LIN {X 0,Y 76.368,Z 462.754,A -85,B 0,C 180,E1 -16863.516,E2 -16863.516} C_VEL
LIN {X 0,Y 76.196,Z 460.368,A -85,B 0,C 180,E1 -16851.651,E2 -16851.651} C_VEL
LIN {X 0,Y 77.548,Z 457.672,A -85,B 0,C 180,E1 -16843.095,E2 -16843.095} C_VEL
LIN {X 0,Y 80.04,Z 454.152,A -85,B 0,C 180,E1 -16835.037,E2 -16835.037} C_VEL
LIN {X 0,Y 84.954,Z 448.19,A -85,B 0,C 180,E1 -16825.255,E2 -16825.255} C_VEL
LIN {X 0,Y 90.817,Z 441.616,A -85,B 0,C 180,E1 -16817.713,E2 -16817.713} C_VEL
LIN {X 0,Y 97.828,Z 433.607,A -85,B 0,C 180,E1 -16811.138,E2 -16811.138} C_VEL
LIN {X 0,Y 105.868,Z 423.896,A -85,B 0,C 180,E1 -16805.487,E2 -16805.487} C_VEL
LIN {X 0,Y 112.858,Z 414.711,A -85,B 0,C 180,E1 -16801.582,E2 -16801.582} C_VEL
LIN {X 0,Y 115.371,Z 410.573,A -85,B 0,C 180,E1 -16799.882,E2 -16799.882} C_VEL
LIN {X 0,Y 118.211,Z 403.586,A -85,B 0,C 180,E1 -16796.713,E2 -16796.713} C_VEL
LIN {X 0,Y 121.079,Z 396.289,A -85,B 0,C 180,E1 -16793.8,E2 -16793.8} C_VEL
LIN {X 0,Y 123.45,Z 391.571,A -85,B 0,C 180,E1 -16792.555,E2 -16792.555} C_VEL
LIN {X 0,Y 130.553,Z 378.137,A -85,B 0,C 180,E1 -16790.263,E2 -16790.263} C_VEL
LIN {X 0,Y 134.162,Z 370.217,A -85,B 0,C 180,E1 -16789.189,E2 -16789.189} C_VEL
LIN {X 0,Y 133.423,Z 370.173,A -85,B 0,C 180,E1 -16788.645,E2 -16788.645} C_VEL
LIN {X 0,Y 123.991,Z 379.977,A -85,B 0,C 180,E1 -16786.279,E2 -16786.279} C_VEL
LIN {X 0,Y 117.805,Z 385.302,A -85,B 0,C 180,E1 -16784.146,E2 -16784.146} C_VEL
LIN {X 0,Y 111.854,Z 389.553,A -85,B 0,C 180,E1 -16781.281,E2 -16781.281} C_VEL
LIN {X 0,Y 106.22,Z 394.346,A -85,B 0,C 180,E1 -16778.946,E2 -16778.946} C_VEL
LIN {X 0,Y 101.258,Z 398.024,A -85,B 0,C 180,E1 -16776.156,E2 -16776.156} C_VEL
LIN {X 0,Y 97.039,Z 400.849,A -85,B 0,C 180,E1 -16772.902,E2 -16772.902} C_VEL
LIN {X 0,Y 90.596,Z 405.763,A -85,B 0,C 180,E1 -16767.741,E2 -16767.741} C_VEL
LIN {X 0,Y 84.281,Z 410.653,A -85,B 0,C 180,E1 -16759.486,E2 -16759.486} C_VEL
LIN {X 0,Y 81.446,Z 413.429,A -85,B 0,C 180,E1 -16755.005,E2 -16755.005} C_VEL
LIN {X 0,Y 79.154,Z 416.279,A -85,B 0,C 180,E1 -16747.655,E2 -16747.655} C_VEL
LIN {X 0,Y 76.953,Z 420.193,A -85,B 0,C 180,E1 -16740.002,E2 -16740.002} C_VEL
LIN {X 0,Y 77.191,Z 424.191,A -85,B 0,C 180,E1 -16729.51,E2 -16729.51} C_VEL
LIN {X 0,Y 79.178,Z 430.201,A -85,B 0,C 180,E1 -16716.459,E2 -16716.459} C_VEL
LIN {X 0,Y 82.647,Z 433.114,A -85,B 0,C 180,E1 -16709.323,E2 -16709.323} C_VEL
LIN {X 0,Y 92.152,Z 437.49,A -85,B 0,C 180,E1 -16698.471,E2 -16698.471} C_VEL
LIN {X 0,Y 91.589,Z 439.223,A -85,B 0,C 180,E1 -16696.801,E2 -16696.801} C_VEL
LIN {X 0,Y 83.49,Z 446.528,A -85,B 0,C 180,E1 -16690.749,E2 -16690.749} C_VEL
LIN {X 0,Y 77.128,Z 452.633,A -85,B 0,C 180,E1 -16683.143,E2 -16683.143} C_VEL
LIN {X 0,Y 72.236,Z 458.21,A -85,B 0,C 180,E1 -16672.903,E2 -16672.903} C_VEL
LIN {X 0,Y 69.917,Z 462.377,A -85,B 0,C 180,E1 -16661.598,E2 -16661.598} C_VEL
LIN {X 0,Y 69.61,Z 463.952,A -85,B 0,C 180,E1 -16655.795,E2 -16655.795} C_VEL
LIN {X 0,Y 69.707,Z 465.196,A -85,B 0,C 180,E1 -16650,E2 -16650} C_VEL
LIN {X 0,Y 69.949,Z 466.704,A -85,B 0,C 180,E1 -16638.408,E2 -16638.408} C_VEL
LIN {X 0,Y 72.306,Z 467.097,A -85,B 0,C 180,E1 -16627.121,E2 -16627.121} C_VEL
LIN {X 0,Y 77.196,Z 466.368,A -85,B 0,C 180,E1 -16616.89,E2 -16616.89} C_VEL
LIN {X 0,Y 84.217,Z 464.543,A -85,B 0,C 180,E1 -16608.117,E2 -16608.117} C_VEL
LIN {X 0,Y 92.984,Z 461.628,A -85,B 0,C 180,E1 -16600.902,E2 -16600.902} C_VEL
LIN {X 0,Y 78.146,Z 461.321,A -85,B 0,C 180,E1 -16559.998,E2 -16559.998} C_VEL
LIN {X 0,Y 82.82,Z 461.492,A -85,B 0,C 180,E1 -16545.25,E2 -16545.25} C_VEL
LIN {X 0,Y 86.083,Z 461.662,A -85,B 0,C 180,E1 -16539.043,E2 -16539.043} C_VEL
LIN {X 0,Y 84.24,Z 462.202,A -85,B 0,C 180,E1 -16536.594,E2 -16536.594} C_VEL
LIN {X 0,Y 76.311,Z 463.737,A -85,B 0,C 180,E1 -16525.983,E2 -16525.983} C_VEL
LIN {X 0,Y 72.236,Z 463.873,A -85,B 0,C 180,E1 -16517.072,E2 -16517.072} C_VEL
LIN {X 0,Y 69.528,Z 463.058,A -85,B 0,C 180,E1 -16506.032,E2 -16506.032} C_VEL
LIN {X 0,Y 68.936,Z 460.88,A -85,B 0,C 180,E1 -16493.425,E2 -16493.425} C_VEL
LIN {X 0,Y 70.739,Z 457.451,A -85,B 0,C 180,E1 -16481.461,E2 -16481.461} C_VEL
LIN {X 0,Y 73.551,Z 453.808,A -85,B 0,C 180,E1 -16472.738,E2 -16472.738} C_VEL
LIN {X 0,Y 79.159,Z 447.606,A -85,B 0,C 180,E1 -16462.215,E2 -16462.215} C_VEL
LIN {X 0,Y 85.499,Z 440.957,A -85,B 0,C 180,E1 -16454.505,E2 -16454.505} C_VEL
LIN {X 0,Y 93.156,Z 432.752,A -85,B 0,C 180,E1 -16447.839,E2 -16447.839} C_VEL
LIN {X 0,Y 100.437,Z 424.367,A -85,B 0,C 180,E1 -16442.946,E2 -16442.946} C_VEL
LIN {X 0,Y 108.34,Z 414.448,A -85,B 0,C 180,E1 -16438.738,E2 -16438.738} C_VEL
LIN {X 0,Y 116.635,Z 402.628,A -85,B 0,C 180,E1 -16435.08,E2 -16435.08} C_VEL
LIN {X 0,Y 123.45,Z 391.571,A -85,B 0,C 180,E1 -16432.555,E2 -16432.555} C_VEL
LIN {X 0,Y 123.693,Z 390.413,A -85,B 0,C 180,E1 -16432.047,E2 -16432.047} C_VEL
LIN {X 0,Y 122.96,Z 389.526,A -85,B 0,C 180,E1 -16431.012,E2 -16431.012} C_VEL
LIN {X 0,Y 120.68,Z 389.525,A -85,B 0,C 180,E1 -16429.342,E2 -16429.342} C_VEL
LIN {X 0,Y 117.78,Z 390.583,A -85,B 0,C 180,E1 -16427.744,E2 -16427.744} C_VEL
LIN {X 0,Y 110.801,Z 394.743,A -85,B 0,C 180,E1 -16424.483,E2 -16424.483} C_VEL
LIN {X 0,Y 103.705,Z 399.598,A -85,B 0,C 180,E1 -16421.335,E2 -16421.335} C_VEL
LIN {X 0,Y 97.384,Z 403.751,A -85,B 0,C 180,E1 -16417.839,E2 -16417.839} C_VEL
LIN {X 0,Y 92.834,Z 406.61,A -85,B 0,C 180,E1 -16414.598,E2 -16414.598} C_VEL
LIN {X 0,Y 86.117,Z 411.175,A -85,B 0,C 180,E1 -16409.32,E2 -16409.32} C_VEL
LIN {X 0,Y 80.97,Z 414.622,A -85,B 0,C 180,E1 -16402.993,E2 -16402.993} C_VEL
LIN {X 0,Y 76.41,Z 418.434,A -85,B 0,C 180,E1 -16396.019,E2 -16396.019} C_VEL
LIN {X 0,Y 74.563,Z 420.264,A -85,B 0,C 180,E1 -16390.868,E2 -16390.868} C_VEL
LIN {X 0,Y 71.362,Z 425.036,A -85,B 0,C 180,E1 -16380.002,E2 -16380.002} C_VEL
LIN {X 0,Y 71.472,Z 428.917,A -85,B 0,C 180,E1 -16368.66,E2 -16368.66} C_VEL
LIN {X 0,Y 72.869,Z 433.562,A -85,B 0,C 180,E1 -16357.309,E2 -16357.309} C_VEL
LIN {X 0,Y 77.582,Z 437.267,A -85,B 0,C 180,E1 -16347.078,E2 -16347.078} C_VEL
LIN {X 0,Y 81.006,Z 438.858,A -85,B 0,C 180,E1 -16342.606,E2 -16342.606} C_VEL
LIN {X 0,Y 84.293,Z 440.47,A -85,B 0,C 180,E1 -16338.623,E2 -16338.623} C_VEL
LIN {X 0,Y 76.372,Z 447.271,A -85,B 0,C 180,E1 -16332.436,E2 -16332.436} C_VEL
LIN {X 0,Y 69.623,Z 453.481,A -85,B 0,C 180,E1 -16323.724,E2 -16323.724} C_VEL
LIN {X 0,Y 64.755,Z 458.82,A -85,B 0,C 180,E1 -16312.325,E2 -16312.325} C_VEL
LIN {X 0,Y 62.925,Z 461.866,A -85,B 0,C 180,E1 -16302.907,E2 -16302.907} C_VEL
LIN {X 0,Y 62.529,Z 463.502,A -85,B 0,C 180,E1 -16296.453,E2 -16296.453} C_VEL
LIN {X 0,Y 62.612,Z 464.805,A -85,B 0,C 180,E1 -16290,E2 -16290} C_VEL
LIN {X 0,Y 62.988,Z 466.428,A -85,B 0,C 180,E1 -16277.106,E2 -16277.106} C_VEL
LIN {X 0,Y 65.766,Z 466.905,A -85,B 0,C 180,E1 -16264.694,E2 -16264.694} C_VEL
LIN {X 0,Y 71.307,Z 466.272,A -85,B 0,C 180,E1 -16253.747,E2 -16253.747} C_VEL
LIN {X 0,Y 79.047,Z 464.579,A -85,B 0,C 180,E1 -16244.661,E2 -16244.661} C_VEL
LIN {X 0,Y 83.577,Z 463.328,A -85,B 0,C 180,E1 -16240.816,E2 -16240.816} C_VEL
LIN {X 0,Y 81.373,Z 463.081,A -85,B 0,C 180,E1 -16237.196,E2 -16237.196} C_VEL
LIN {X 0,Y 71.135,Z 462.672,A -85,B 0,C 180,E1 -16199.998,E2 -16199.998} C_VEL
LIN {X 0,Y 76.059,Z 462.669,A -85,B 0,C 180,E1 -16183.905,E2 -16183.905} C_VEL
LIN {X 0,Y 77.863,Z 462.842,A -85,B 0,C 180,E1 -16178.834,E2 -16178.834} C_VEL
LIN {X 0,Y 71.168,Z 463.889,A -85,B 0,C 180,E1 -16170.41,E2 -16170.41} C_VEL
LIN {X 0,Y 65.431,Z 464.015,A -85,B 0,C 180,E1 -16158.753,E2 -16158.753} C_VEL
LIN {X 0,Y 62.714,Z 463.261,A -85,B 0,C 180,E1 -16148.327,E2 -16148.327} C_VEL
LIN {X 0,Y 61.773,Z 461.123,A -85,B 0,C 180,E1 -16134.466,E2 -16134.466} C_VEL
LIN {X 0,Y 64.067,Z 457.031,A -85,B 0,C 180,E1 -16119.137,E2 -16119.137} C_VEL
LIN {X 0,Y 67.197,Z 453.432,A -85,B 0,C 180,E1 -16110,E2 -16110} C_VEL
LIN {X 0,Y 73.42,Z 447.159,A -85,B 0,C 180,E1 -16098.963,E2 -16098.963} C_VEL
LIN {X 0,Y 80.518,Z 440.248,A -85,B 0,C 180,E1 -16090.894,E2 -16090.894} C_VEL
LIN {X 0,Y 88.791,Z 431.855,A -85,B 0,C 180,E1 -16084.193,E2 -16084.193} C_VEL
LIN {X 0,Y 97.541,Z 422.163,A -85,B 0,C 180,E1 -16078.854,E2 -16078.854} C_VEL
LIN {X 0,Y 106.362,Z 411.255,A -85,B 0,C 180,E1 -16074.678,E2 -16074.678} C_VEL
LIN {X 0,Y 114.373,Z 399.873,A -85,B 0,C 180,E1 -16071.526,E2 -16071.526} C_VEL
LIN {X 0,Y 122.079,Z 387.208,A -85,B 0,C 180,E1 -16068.968,E2 -16068.968} C_VEL
LIN {X 0,Y 122.246,Z 385.942,A -85,B 0,C 180,E1 -16068.365,E2 -16068.365} C_VEL
LIN {X 0,Y 116.352,Z 390.487,A -85,B 0,C 180,E1 -16066.457,E2 -16066.457} C_VEL
LIN {X 0,Y 111.037,Z 394.055,A -85,B 0,C 180,E1 -16064.128,E2 -16064.128} C_VEL
LIN {X 0,Y 103.705,Z 399.598,A -85,B 0,C 180,E1 -16061.335,E2 -16061.335} C_VEL
LIN {X 0,Y 98.192,Z 403.895,A -85,B 0,C 180,E1 -16059.172,E2 -16059.172} C_VEL
LIN {X 0,Y 86.954,Z 412.786,A -85,B 0,C 180,E1 -16054.923,E2 -16054.923} C_VEL
LIN {X 0,Y 83.121,Z 415.36,A -85,B 0,C 180,E1 -16052.518,E2 -16052.518} C_VEL
LIN {X 0,Y 81.981,Z 416.062,A -85,B 0,C 180,E1 -16051.537,E2 -16051.537} C_VEL
LIN {X 0,Y 75.939,Z 419.737,A -85,B 0,C 180,E1 -16044.614,E2 -16044.614} C_VEL
LIN {X 0,Y 71.207,Z 423.205,A -85,B 0,C 180,E1 -16037.225,E2 -16037.225} C_VEL
LIN {X 0,Y 69.088,Z 425.046,A -85,B 0,C 180,E1 -16031.741,E2 -16031.741} C_VEL
LIN {X 0,Y 65.659,Z 429.569,A -85,B 0,C 180,E1 -16020.002,E2 -16020.002} C_VEL
LIN {X 0,Y 65.52,Z 432.275,A -85,B 0,C 180,E1 -16010.743,E2 -16010.743} C_VEL
LIN {X 0,Y 67.295,Z 437.714,A -85,B 0,C 180,E1 -15995.31,E2 -15995.31} C_VEL
LIN {X 0,Y 74.24,Z 441.892,A -85,B 0,C 180,E1 -15982.129,E2 -15982.129} C_VEL
LIN {X 0,Y 75.152,Z 442.251,A -85,B 0,C 180,E1 -15981.015,E2 -15981.015} C_VEL
LIN {X 0,Y 74.569,Z 443.749,A -85,B 0,C 180,E1 -15978.937,E2 -15978.937} C_VEL
LIN {X 0,Y 67.66,Z 449.413,A -85,B 0,C 180,E1 -15972.467,E2 -15972.467} C_VEL
LIN {X 0,Y 60.672,Z 455.626,A -85,B 0,C 180,E1 -15961.417,E2 -15961.417} C_VEL
LIN {X 0,Y 56.532,Z 460.378,A -85,B 0,C 180,E1 -15948.107,E2 -15948.107} C_VEL
LIN {X 0,Y 55.45,Z 463.046,A -85,B 0,C 180,E1 -15937.282,E2 -15937.282} C_VEL
LIN {X 0,Y 55.507,Z 464.411,A -85,B 0,C 180,E1 -15930,E2 -15930} C_VEL
LIN {X 0,Y 55.478,Z 465.428,A -85,B 0,C 180,E1 -15922.722,E2 -15922.722} C_VEL
LIN {X 0,Y 57.334,Z 466.545,A -85,B 0,C 180,E1 -15908.424,E2 -15908.424} C_VEL
LIN {X 0,Y 62.236,Z 466.565,A -85,B 0,C 180,E1 -15895.624,E2 -15895.624} C_VEL
LIN {X 0,Y 70.132,Z 465.439,A -85,B 0,C 180,E1 -15884.543,E2 -15884.543} C_VEL
LIN {X 0,Y 74.205,Z 464.618,A -85,B 0,C 180,E1 -15880.74,E2 -15880.74} C_VEL
LIN {X 0,Y 72.274,Z 464.257,A -85,B 0,C 180,E1 -15875.691,E2 -15875.691} C_VEL
LIN {X 0,Y 65.156,Z 463.678,A -85,B 0,C 180,E1 -15833.806,E2 -15833.806} C_VEL
LIN {X 0,Y 69.294,Z 463.577,A -85,B 0,C 180,E1 -15822.284,E2 -15822.284} C_VEL
LIN {X 0,Y 69.917,Z 463.604,A -85,B 0,C 180,E1 -15820.416,E2 -15820.416} C_VEL
LIN {X 0,Y 68.306,Z 463.862,A -85,B 0,C 180,E1 -15817.822,E2 -15817.822} C_VEL
LIN {X 0,Y 60.284,Z 464.28,A -85,B 0,C 180,E1 -15804.694,E2 -15804.694} C_VEL
LIN {X 0,Y 55.656,Z 463.224,A -85,B 0,C 180,E1 -15789.152,E2 -15789.152} C_VEL
LIN {X 0,Y 54.654,Z 461.369,A -85,B 0,C 180,E1 -15775.819,E2 -15775.819} C_VEL
LIN {X 0,Y 56.877,Z 457.36,A -85,B 0,C 180,E1 -15758.675,E2 -15758.675} C_VEL
LIN {X 0,Y 61.019,Z 453.04,A -85,B 0,C 180,E1 -15746.699,E2 -15746.699} C_VEL
LIN {X 0,Y 66.104,Z 448.307,A -85,B 0,C 180,E1 -15737.723,E2 -15737.723} C_VEL
LIN {X 0,Y 73.546,Z 441.623,A -85,B 0,C 180,E1 -15729.001,E2 -15729.001} C_VEL
LIN {X 0,Y 82.156,Z 433.491,A -85,B 0,C 180,E1 -15721.934,E2 -15721.934} C_VEL
LIN {X 0,Y 91.523,Z 423.833,A -85,B 0,C 180,E1 -15716.34,E2 -15716.34} C_VEL
LIN {X 0,Y 100.423,Z 413.508,A -85,B 0,C 180,E1 -15712.24,E2 -15712.24} C_VEL
LIN {X 0,Y 108.874,Z 402.258,A -85,B 0,C 180,E1 -15709.042,E2 -15709.042} C_VEL
LIN {X 0,Y 110.997,Z 399.206,A -85,B 0,C 180,E1 -15708.331,E2 -15708.331} C_VEL
LIN {X 0,Y 111.248,Z 397.843,A -85,B 0,C 180,E1 -15707.482,E2 -15707.482} C_VEL
LIN {X 0,Y 109.367,Z 399.017,A -85,B 0,C 180,E1 -15706.717,E2 -15706.717} C_VEL
LIN {X 0,Y 102.458,Z 403.878,A -85,B 0,C 180,E1 -15704.4,E2 -15704.4} C_VEL
LIN {X 0,Y 95.928,Z 407.841,A -85,B 0,C 180,E1 -15701.254,E2 -15701.254} C_VEL
LIN {X 0,Y 88.475,Z 412.197,A -85,B 0,C 180,E1 -15696.569,E2 -15696.569} C_VEL
LIN {X 0,Y 84.862,Z 414.371,A -85,B 0,C 180,E1 -15694.089,E2 -15694.089} C_VEL
LIN {X 0,Y 81.981,Z 416.062,A -85,B 0,C 180,E1 -15691.537,E2 -15691.537} C_VEL
LIN {X 0,Y 78.449,Z 418.43,A -85,B 0,C 180,E1 -15688.587,E2 -15688.587} C_VEL
LIN {X 0,Y 66.301,Z 427.363,A -85,B 0,C 180,E1 -15678.414,E2 -15678.414} C_VEL
LIN {X 0,Y 63.817,Z 429.257,A -85,B 0,C 180,E1 -15674.051,E2 -15674.051} C_VEL
LIN {X 0,Y 59.784,Z 433.842,A -85,B 0,C 180,E1 -15660.002,E2 -15660.002} C_VEL
LIN {X 0,Y 59.452,Z 436.535,A -85,B 0,C 180,E1 -15649.788,E2 -15649.788} C_VEL
LIN {X 0,Y 60.029,Z 439.741,A -85,B 0,C 180,E1 -15639.44,E2 -15639.44} C_VEL
LIN {X 0,Y 67.19,Z 445.033,A -85,B 0,C 180,E1 -15621.129,E2 -15621.129} C_VEL
LIN {X 0,Y 58.279,Z 451.919,A -85,B 0,C 180,E1 -15611.549,E2 -15611.549} C_VEL
LIN {X 0,Y 51.8,Z 457.526,A -85,B 0,C 180,E1 -15598.351,E2 -15598.351} C_VEL
LIN {X 0,Y 49.121,Z 460.826,A -85,B 0,C 180,E1 -15586.627,E2 -15586.627} C_VEL
LIN {X 0,Y 48.382,Z 462.584,A -85,B 0,C 180,E1 -15578.352,E2 -15578.352} C_VEL
LIN {X 0,Y 48.421,Z 464.003,A -85,B 0,C 180,E1 -15570,E2 -15570} C_VEL
LIN {X 0,Y 48.428,Z 465.045,A -85,B 0,C 180,E1 -15561.656,E2 -15561.656} C_VEL
LIN {X 0,Y 50.747,Z 466.261,A -85,B 0,C 180,E1 -15545.451,E2 -15545.451} C_VEL
LIN {X 0,Y 56.472,Z 466.41,A -85,B 0,C 180,E1 -15531.519,E2 -15531.519} C_VEL
LIN {X 0,Y 64.794,Z 465.508,A -85,B 0,C 180,E1 -15520.6,E2 -15520.6} C_VEL
LIN {X 0,Y 65.729,Z 465.194,A -85,B 0,C 180,E1 -15517.936,E2 -15517.936} C_VEL
LIN {X 0,Y 58.132,Z 464.423,A -85,B 0,C 180,E1 -15473.054,E2 -15473.054} C_VEL
LIN {X 0,Y 59.955,Z 464.32,A -85,B 0,C 180,E1 -15466.439,E2 -15466.439} C_VEL
LIN {X 0,Y 61.232,Z 464.317,A -85,B 0,C 180,E1 -15459.857,E2 -15459.857} C_VEL
LIN {X 0,Y 54.408,Z 464.457,A -85,B 0,C 180,E1 -15448.887,E2 -15448.887} C_VEL
LIN {X 0,Y 49.492,Z 463.647,A -85,B 0,C 180,E1 -15434.76,E2 -15434.76} C_VEL
LIN {X 0,Y 47.557,Z 461.589,A -85,B 0,C 180,E1 -15417.535,E2 -15417.535} C_VEL
LIN {X 0,Y 48.749,Z 458.73,A -85,B 0,C 180,E1 -15402.489,E2 -15402.489} C_VEL
LIN {X 0,Y 52.04,Z 455.302,A -85,B 0,C 180,E1 -15390,E2 -15390} C_VEL
LIN {X 0,Y 58.831,Z 449.438,A -85,B 0,C 180,E1 -15376.177,E2 -15376.177} C_VEL
LIN {X 0,Y 66.648,Z 442.987,A -85,B 0,C 180,E1 -15366.707,E2 -15366.707} C_VEL
LIN {X 0,Y 75.693,Z 435.109,A -85,B 0,C 180,E1 -15359.292,E2 -15359.292} C_VEL
LIN {X 0,Y 84.195,Z 427.056,A -85,B 0,C 180,E1 -15354.246,E2 -15354.246} C_VEL
LIN {X 0,Y 93.131,Z 417.524,A -85,B 0,C 180,E1 -15350.101,E2 -15350.101} C_VEL
LIN {X 0,Y 99.342,Z 410.162,A -85,B 0,C 180,E1 -15347.772,E2 -15347.772} C_VEL
LIN {X 0,Y 99.514,Z 409.158,A -85,B 0,C 180,E1 -15346.891,E2 -15346.891} C_VEL
LIN {X 0,Y 92.083,Z 413.127,A -85,B 0,C 180,E1 -15343.387,E2 -15343.387} C_VEL
LIN {X 0,Y 81.519,Z 418.843,A -85,B 0,C 180,E1 -15337.123,E2 -15337.123} C_VEL
LIN {X 0,Y 70.406,Z 424.828,A -85,B 0,C 180,E1 -15326.052,E2 -15326.052} C_VEL
LIN {X 0,Y 63.817,Z 429.257,A -85,B 0,C 180,E1 -15314.051,E2 -15314.051} C_VEL
LIN {X 0,Y 61.647,Z 431.159,A -85,B 0,C 180,E1 -15309.357,E2 -15309.357} C_VEL
LIN {X 0,Y 57.393,Z 435.16,A -85,B 0,C 180,E1 -15301.653,E2 -15301.653} C_VEL
LIN {X 0,Y 54.449,Z 438.384,A -85,B 0,C 180,E1 -15294.804,E2 -15294.804} C_VEL
LIN {X 0,Y 53.274,Z 440.398,A -85,B 0,C 180,E1 -15289.006,E2 -15289.006} C_VEL
LIN {X 0,Y 53.192,Z 440.973,A -85,B 0,C 180,E1 -15286.974,E2 -15286.974} C_VEL
LIN {X 0,Y 56.079,Z 445.201,A -85,B 0,C 180,E1 -15269.917,E2 -15269.917} C_VEL
LIN {X 0,Y 58.874,Z 446.826,A -85,B 0,C 180,E1 -15263.356,E2 -15263.356} C_VEL
LIN {X 0,Y 55.501,Z 449.464,A -85,B 0,C 180,E1 -15259.444,E2 -15259.444} C_VEL
LIN {X 0,Y 47.232,Z 455.578,A -85,B 0,C 180,E1 -15246.526,E2 -15246.526} C_VEL
LIN {X 0,Y 42.321,Z 460.243,A -85,B 0,C 180,E1 -15229.398,E2 -15229.398} C_VEL
LIN {X 0,Y 41.353,Z 462.056,A -85,B 0,C 180,E1 -15219.785,E2 -15219.785} C_VEL
LIN {X 0,Y 41.315,Z 463.53,A -85,B 0,C 180,E1 -15210,E2 -15210} C_VEL
LIN {X 0,Y 41.392,Z 464.634,A -85,B 0,C 180,E1 -15200.224,E2 -15200.224} C_VEL
LIN {X 0,Y 44.347,Z 465.978,A -85,B 0,C 180,E1 -15181.612,E2 -15181.612} C_VEL
LIN {X 0,Y 51.054,Z 466.255,A -85,B 0,C 180,E1 -15166.505,E2 -15166.505} C_VEL
LIN {X 0,Y 55.467,Z 466.004,A -85,B 0,C 180,E1 -15160.515,E2 -15160.515} C_VEL
LIN {X 0,Y 57.368,Z 465.762,A -85,B 0,C 180,E1 -15157.77,E2 -15157.77} C_VEL
LIN {X 0,Y 51.069,Z 464.892,A -85,B 0,C 180,E1 -15112.087,E2 -15112.087} C_VEL
LIN {X 0,Y 53.071,Z 464.732,A -85,B 0,C 180,E1 -15104.639,E2 -15104.639} C_VEL
LIN {X 0,Y 52.388,Z 464.709,A -85,B 0,C 180,E1 -15099.896,E2 -15099.896} C_VEL
LIN {X 0,Y 47.803,Z 464.569,A -85,B 0,C 180,E1 -15091.899,E2 -15091.899} C_VEL
LIN {X 0,Y 41.686,Z 463.204,A -85,B 0,C 180,E1 -15072.406,E2 -15072.406} C_VEL
LIN {X 0,Y 40.504,Z 461.803,A -85,B 0,C 180,E1 -15059.816,E2 -15059.816} C_VEL
LIN {X 0,Y 41.991,Z 458.478,A -85,B 0,C 180,E1 -15039.635,E2 -15039.635} C_VEL
LIN {X 0,Y 45.925,Z 454.887,A -85,B 0,C 180,E1 -15025.612,E2 -15025.612} C_VEL
LIN {X 0,Y 51.582,Z 450.543,A -85,B 0,C 180,E1 -15014.187,E2 -15014.187} C_VEL
LIN {X 0,Y 58.577,Z 445.229,A -85,B 0,C 180,E1 -15005.17,E2 -15005.17} C_VEL
LIN {X 0,Y 67.98,Z 437.785,A -85,B 0,C 180,E1 -14997.128,E2 -14997.128} C_VEL
LIN {X 0,Y 78.316,Z 428.749,A -85,B 0,C 180,E1 -14991.084,E2 -14991.084} C_VEL
LIN {X 0,Y 87.44,Z 419.673,A -85,B 0,C 180,E1 -14987.07,E2 -14987.07} C_VEL
LIN {X 0,Y 88.191,Z 418.229,A -85,B 0,C 180,E1 -14985.828,E2 -14985.828} C_VEL
LIN {X 0,Y 77.13,Z 423.642,A -85,B 0,C 180,E1 -14979.633,E2 -14979.633} C_VEL
LIN {X 0,Y 67.839,Z 428.045,A -85,B 0,C 180,E1 -14971.2,E2 -14971.2} C_VEL
LIN {X 0,Y 60.123,Z 432.201,A -85,B 0,C 180,E1 -14959.997,E2 -14959.997} C_VEL
LIN {X 0,Y 53.738,Z 437.87,A -85,B 0,C 180,E1 -14940.002,E2 -14940.002} C_VEL
LIN {X 0,Y 53.333,Z 439.545,A -85,B 0,C 180,E1 -14932.43,E2 -14932.43} C_VEL
LIN {X 0,Y 53.192,Z 440.973,A -85,B 0,C 180,E1 -14926.974,E2 -14926.974} C_VEL
LIN {X 0,Y 53.125,Z 443.11,A -85,B 0,C 180,E1 -14919.775,E2 -14919.775} C_VEL
LIN {X 0,Y 52.713,Z 445.096,A -85,B 0,C 180,E1 -14914.172,E2 -14914.172} C_VEL
LIN {X 0,Y 51.578,Z 447.285,A -85,B 0,C 180,E1 -14908.893,E2 -14908.893} C_VEL
LIN {X 0,Y 49.94,Z 449.033,A -85,B 0,C 180,E1 -14905.254,E2 -14905.254} C_VEL
LIN {X 0,Y 48.476,Z 450.307,A -85,B 0,C 180,E1 -14902.719,E2 -14902.719} C_VEL
LIN {X 0,Y 39.807,Z 456.16,A -85,B 0,C 180,E1 -14888.165,E2 -14888.165} C_VEL
LIN {X 0,Y 35.667,Z 459.63,A -85,B 0,C 180,E1 -14873.209,E2 -14873.209} C_VEL
LIN {X 0,Y 34.226,Z 463.056,A -85,B 0,C 180,E1 -14850,E2 -14850} C_VEL
LIN {X 0,Y 34.407,Z 464.222,A -85,B 0,C 180,E1 -14838.214,E2 -14838.214} C_VEL
LIN {X 0,Y 38.196,Z 465.688,A -85,B 0,C 180,E1 -14816.496,E2 -14816.496} C_VEL
LIN {X 0,Y 46.118,Z 466.098,A -85,B 0,C 180,E1 -14800.362,E2 -14800.362} C_VEL
LIN {X 0,Y 48.164,Z 465.952,A -85,B 0,C 180,E1 -14795.706,E2 -14795.706} C_VEL
LIN {X 0,Y 44.027,Z 465.08,A -85,B 0,C 180,E1 -14750.812,E2 -14750.812} C_VEL
LIN {X 0,Y 45.595,Z 464.92,A -85,B 0,C 180,E1 -14744.348,E2 -14744.348} C_VEL
LIN {X 0,Y 44.462,Z 464.836,A -85,B 0,C 180,E1 -14741.514,E2 -14741.514} C_VEL
LIN {X 0,Y 37.302,Z 464.009,A -85,B 0,C 180,E1 -14725.578,E2 -14725.578} C_VEL
LIN {X 0,Y 33.518,Z 461.997,A -85,B 0,C 180,E1 -14702.99,E2 -14702.99} C_VEL
LIN {X 0,Y 35.332,Z 458.216,A -85,B 0,C 180,E1 -14675.932,E2 -14675.932} C_VEL
LIN {X 0,Y 40.148,Z 454.471,A -85,B 0,C 180,E1 -14659.918,E2 -14659.918} C_VEL
LIN {X 0,Y 46.834,Z 449.908,A -85,B 0,C 180,E1 -14647.83,E2 -14647.83} C_VEL
LIN {X 0,Y 57.518,Z 442.479,A -85,B 0,C 180,E1 -14636.643,E2 -14636.643} C_VEL
LIN {X 0,Y 67.959,Z 434.414,A -85,B 0,C 180,E1 -14629.733,E2 -14629.733} C_VEL
LIN {X 0,Y 75.887,Z 427.648,A -85,B 0,C 180,E1 -14626.006,E2 -14626.006} C_VEL
LIN {X 0,Y 76.439,Z 426.655,A -85,B 0,C 180,E1 -14624.821,E2 -14624.821} C_VEL
LIN {X 0,Y 58.395,Z 434.353,A -85,B 0,C 180,E1 -14608.78,E2 -14608.78} C_VEL
LIN {X 0,Y 51.511,Z 438.053,A -85,B 0,C 180,E1 -14595.838,E2 -14595.838} C_VEL
LIN {X 0,Y 46.856,Z 444.055,A -85,B 0,C 180,E1 -14567.94,E2 -14567.94} C_VEL
LIN {X 0,Y 50.54,Z 448.533,A -85,B 0,C 180,E1 -14546.207,E2 -14546.207} C_VEL
LIN {X 0,Y 49.94,Z 449.033,A -85,B 0,C 180,E1 -14545.254,E2 -14545.254} C_VEL
LIN {X 0,Y 47.614,Z 450.723,A -85,B 0,C 180,E1 -14542.143,E2 -14542.143} C_VEL
LIN {X 0,Y 43.348,Z 453.054,A -85,B 0,C 180,E1 -14537.923,E2 -14537.923} C_VEL
LIN {X 0,Y 32.518,Z 457.53,A -85,B 0,C 180,E1 -14526.021,E2 -14526.021} C_VEL
LIN {X 0,Y 29.076,Z 459.218,A -85,B 0,C 180,E1 -14517.349,E2 -14517.349} C_VEL
LIN {X 0,Y 28.369,Z 459.728,A -85,B 0,C 180,E1 -14513.761,E2 -14513.761} C_VEL
LIN {X 0,Y 27.109,Z 462.562,A -85,B 0,C 180,E1 -14490,E2 -14490} C_VEL
LIN {X 0,Y 27.466,Z 463.794,A -85,B 0,C 180,E1 -14475.175,E2 -14475.175} C_VEL
LIN {X 0,Y 32.467,Z 465.398,A -85,B 0,C 180,E1 -14449.504,E2 -14449.504} C_VEL
LIN {X 0,Y 39.252,Z 465.845,A -85,B 0,C 180,E1 -14436.252,E2 -14436.252} C_VEL
LIN {X 0,Y 39.02,Z 465.797,A -85,B 0,C 180,E1 -14432.703,E2 -14432.703} C_VEL
LIN {X 0,Y 37.016,Z 464.97,A -85,B 0,C 180,E1 -14389.052,E2 -14389.052} C_VEL
LIN {X 0,Y 36.565,Z 464.786,A -85,B 0,C 180,E1 -14383.95,E2 -14383.95} C_VEL
LIN {X 0,Y 31.596,Z 464.101,A -85,B 0,C 180,E1 -14372.842,E2 -14372.842} C_VEL
LIN {X 0,Y 26.687,Z 462.185,A -85,B 0,C 180,E1 -14347.802,E2 -14347.802} C_VEL
LIN {X 0,Y 28.183,Z 458.456,A -85,B 0,C 180,E1 -14313.995,E2 -14313.995} C_VEL
LIN {X 0,Y 34.914,Z 454.019,A -85,B 0,C 180,E1 -14292.425,E2 -14292.425} C_VEL
LIN {X 0,Y 45.465,Z 447.61,A -85,B 0,C 180,E1 -14277.246,E2 -14277.246} C_VEL
LIN {X 0,Y 55.907,Z 440.73,A -85,B 0,C 180,E1 -14268.964,E2 -14268.964} C_VEL
LIN {X 0,Y 64.954,Z 434.003,A -85,B 0,C 180,E1 -14264.189,E2 -14264.189} C_VEL
LIN {X 0,Y 64.14,Z 434.012,A -85,B 0,C 180,E1 -14262.773,E2 -14262.773} C_VEL
LIN {X 0,Y 49.441,Z 439.821,A -85,B 0,C 180,E1 -14246.146,E2 -14246.146} C_VEL
LIN {X 0,Y 40.491,Z 446.786,A -85,B 0,C 180,E1 -14210.008,E2 -14210.008} C_VEL
LIN {X 0,Y 42.34,Z 450.139,A -85,B 0,C 180,E1 -14190.138,E2 -14190.138} C_VEL
LIN {X 0,Y 41.81,Z 451.027,A -85,B 0,C 180,E1 -14187.19,E2 -14187.19} C_VEL
LIN {X 0,Y 32.414,Z 456.696,A -85,B 0,C 180,E1 -14170.576,E2 -14170.576} C_VEL
LIN {X 0,Y 28.369,Z 459.728,A -85,B 0,C 180,E1 -14153.761,E2 -14153.761} C_VEL
LIN {X 0,Y 27.109,Z 460.767,A -85,B 0,C 180,E1 -14146.341,E2 -14146.341} C_VEL
LIN {X 0,Y 25.686,Z 461.638,A -85,B 0,C 180,E1 -14138.578,E2 -14138.578} C_VEL
LIN {X 0,Y 23.231,Z 462.981,A -85,B 0,C 180,E1 -14121.036,E2 -14121.036} C_VEL
LIN {X 0,Y 23.95,Z 464.477,A -85,B 0,C 180,E1 -14091.363,E2 -14091.363} C_VEL
LIN {X 0,Y 25.995,Z 464.841,A -85,B 0,C 180,E1 -14083.391,E2 -14083.391} C_VEL
LIN {X 0,Y 29.384,Z 465.256,A -85,B 0,C 180,E1 -14075.775,E2 -14075.775} C_VEL
LIN {X 0,Y 30.67,Z 465.345,A -85,B 0,C 180,E1 -14070.608,E2 -14070.608} C_VEL
LIN {X 0,Y 28.426,Z 464.815,A -85,B 0,C 180,E1 -14039.996,E2 -14039.996} C_VEL
LIN {X 0,Y 28.773,Z 464.534,A -85,B 0,C 180,E1 -14027.696,E2 -14027.696} C_VEL
LIN {X 0,Y 20.011,Z 462.282,A -85,B 0,C 180,E1 -13994.621,E2 -13994.621} C_VEL
LIN {X 0,Y 21.088,Z 458.692,A -85,B 0,C 180,E1 -13950.7,E2 -13950.7} C_VEL
LIN {X 0,Y 27.768,Z 454.894,A -85,B 0,C 180,E1 -13927.688,E2 -13927.688} C_VEL
LIN {X 0,Y 39.389,Z 448.691,A -85,B 0,C 180,E1 -13911.355,E2 -13911.355} C_VEL
LIN {X 0,Y 51.744,Z 441.232,A -85,B 0,C 180,E1 -13902.778,E2 -13902.778} C_VEL
LIN {X 0,Y 53.051,Z 440.223,A -85,B 0,C 180,E1 -13901.485,E2 -13901.485} C_VEL
LIN {X 0,Y 39.377,Z 445.317,A -85,B 0,C 180,E1 -13880.917,E2 -13880.917} C_VEL
LIN {X 0,Y 34.579,Z 448.407,A -85,B 0,C 180,E1 -13860.004,E2 -13860.004} C_VEL
LIN {X 0,Y 34.498,Z 451.573,A -85,B 0,C 180,E1 -13835.96,E2 -13835.96} C_VEL
LIN {X 0,Y 33.96,Z 452.567,A -85,B 0,C 180,E1 -13831.374,E2 -13831.374} C_VEL
LIN {X 0,Y 23.217,Z 458.354,A -85,B 0,C 180,E1 -13807.26,E2 -13807.26} C_VEL
LIN {X 0,Y 20.599,Z 460.381,A -85,B 0,C 180,E1 -13789.948,E2 -13789.948} C_VEL
LIN {X 0,Y 19.996,Z 462.066,A -85,B 0,C 180,E1 -13770,E2 -13770} C_VEL
LIN {X 0,Y 20.667,Z 463.369,A -85,B 0,C 180,E1 -13750.12,E2 -13750.12} C_VEL
LIN {X 0,Y 25.995,Z 464.841,A -85,B 0,C 180,E1 -13723.391,E2 -13723.391} C_VEL
LIN {X 0,Y 26.328,Z 464.928,A -85,B 0,C 180,E1 -13720.13,E2 -13720.13} C_VEL
LIN {X 0,Y 25.388,Z 464.877,A -85,B 0,C 180,E1 -13714.439,E2 -13714.439} C_VEL
LIN {X 0,Y 21.429,Z 464.41,A -85,B 0,C 180,E1 -13696.894,E2 -13696.894} C_VEL
LIN {X 0,Y 21.321,Z 464.169,A -85,B 0,C 180,E1 -13679.994,E2 -13679.994} C_VEL
LIN {X 0,Y 21.184,Z 464.034,A -85,B 0,C 180,E1 -13674.428,E2 -13674.428} C_VEL
LIN {X 0,Y 14.266,Z 462.507,A -85,B 0,C 180,E1 -13650.475,E2 -13650.475} C_VEL
LIN {X 0,Y 14.139,Z 458.883,A -85,B 0,C 180,E1 -13583.892,E2 -13583.892} C_VEL
LIN {X 0,Y 20.896,Z 455.752,A -85,B 0,C 180,E1 -13559.701,E2 -13559.701} C_VEL
LIN {X 0,Y 30.495,Z 451.421,A -85,B 0,C 180,E1 -13546.259,E2 -13546.259} C_VEL
LIN {X 0,Y 39.829,Z 446.605,A -85,B 0,C 180,E1 -13539.484,E2 -13539.484} C_VEL
LIN {X 0,Y 39.018,Z 446.521,A -85,B 0,C 180,E1 -13535.696,E2 -13535.696} C_VEL
LIN {X 0,Y 27.861,Z 451.398,A -85,B 0,C 180,E1 -13500.005,E2 -13500.005} C_VEL
LIN {X 0,Y 27.348,Z 453.179,A -85,B 0,C 180,E1 -13481.893,E2 -13481.893} C_VEL
LIN {X 0,Y 25.732,Z 454.231,A -85,B 0,C 180,E1 -13477.194,E2 -13477.194} C_VEL
LIN {X 0,Y 15.814,Z 458.765,A -85,B 0,C 180,E1 -13451.806,E2 -13451.806} C_VEL
LIN {X 0,Y 12.897,Z 461.555,A -85,B 0,C 180,E1 -13410,E2 -13410} C_VEL
LIN {X 0,Y 14.192,Z 462.893,A -85,B 0,C 180,E1 -13380.317,E2 -13380.317} C_VEL
LIN {X 0,Y 20.414,Z 464.313,A -85,B 0,C 180,E1 -13352.454,E2 -13352.454} C_VEL
LIN {X 0,Y 22.05,Z 464.514,A -85,B 0,C 180,E1 -13344.062,E2 -13344.062} C_VEL
LIN {X 0,Y 21.429,Z 464.41,A -85,B 0,C 180,E1 -13336.894,E2 -13336.894} C_VEL
LIN {X 0,Y 20.414,Z 464.253,A -85,B 0,C 180,E1 -13331.231,E2 -13331.231} C_VEL
LIN {X 0,Y 18.126,Z 463.91,A -85,B 0,C 180,E1 -13325.321,E2 -13325.321} C_VEL
LIN {X 0,Y 14.098,Z 463.188,A -85,B 0,C 180,E1 -13318.103,E2 -13318.103} C_VEL
LIN {X 0,Y 4.958,Z 460.881,A -85,B 0,C 180,E1 -13267.837,E2 -13267.837} C_VEL
LIN {X 0,Y 4.858,Z 460.632,A -85,B 0,C 180,E1 -13258.944,E2 -13258.944} C_VEL
LIN {X 0,Y 11.27,Z 457.815,A -85,B 0,C 180,E1 -13191.422,E2 -13191.422} C_VEL
LIN {X 0,Y 21.714,Z 453.97,A -85,B 0,C 180,E1 -13177.124,E2 -13177.124} C_VEL
LIN {X 0,Y 25.592,Z 452.347,A -85,B 0,C 180,E1 -13174.527,E2 -13174.527} C_VEL
LIN {X 0,Y 27.454,Z 451.421,A -85,B 0,C 180,E1 -13170.801,E2 -13170.801} C_VEL
LIN {X 0,Y 20.712,Z 454.473,A -85,B 0,C 180,E1 -13134.918,E2 -13134.918} C_VEL
LIN {X 0,Y 17.926,Z 455.749,A -85,B 0,C 180,E1 -13128.18,E2 -13128.18} C_VEL
LIN {X 0,Y 8.68,Z 459.147,A -85,B 0,C 180,E1 -13104.062,E2 -13104.062} C_VEL
LIN {X 0,Y 5.786,Z 460.965,A -85,B 0,C 180,E1 -13050,E2 -13050} C_VEL
LIN {X 0,Y 8.745,Z 462.374,A -85,B 0,C 180,E1 -12996.517,E2 -12996.517} C_VEL
LIN {X 0,Y 14.155,Z 463.356,A -85,B 0,C 180,E1 -12970.587,E2 -12970.587} C_VEL
LIN {X 0,Y 10.416,Z 462.654,A -85,B 0,C 180,E1 -12959.988,E2 -12959.988} C_VEL
LIN {X 0,Y 4.858,Z 460.632,A -85,B 0,C 180,E1 -12898.944,E2 -12898.944} C_VEL
LIN {X 0,Y 4.773,Z 460.055,A -85,B 0,C 180,E1 -12868.95,E2 -12868.95} C_VEL
LIN {X 0,Y 5.567,Z 459.188,A -85,B 0,C 180,E1 -12825.363,E2 -12825.363} C_VEL
LIN {X 0,Y 9.818,Z 457.748,A -85,B 0,C 180,E1 -12790.805,E2 -12790.805} C_VEL
LIN {X 0,Y 12.547,Z 456.914,A -85,B 0,C 180,E1 -12787.517,E2 -12787.517} C_VEL
LIN {X 0,Y 14.105,Z 456.336,A -85,B 0,C 180,E1 -12790.053,E2 -12790.053} C_VEL
LIN {X 0,Y 14.365,Z 456.225,A -85,B 0,C 180,E1 -12791.91,E2 -12791.91} C_VEL
LIN {X 0,Y 14.105,Z 458.214,A -85,B 0,C 180,E1 -12784.775,E2 -12784.775} C_VEL
LIN {X 0,Y 14.105,Z 600,A -85,B 0,C 180,E1 -12784.775,E2 -12784.775} C_VEL
LIN {X 0,Y 14.105,Z 600,A -85,B 0,C 180,E1 -12784.775,E2 -12784.775}

QRS_NEXT_CUT()

QRS_NEXT()
QRS_HOME()

END
